{attribute 'qualified_only'}
VAR_GLOBAL
END_VAR

(* stored: Version 1.1.0.1, ProductVersion 3.1.4024.11
   GVL GVLtest10: Id {85e8af4e-6d09-4018-8968-4c5c590b6078} *)
